// Mitsubishi GX Works2 project: 0624(BKRST_일괄리셋)   PLC: Q02/Q02H

PROGRAM MAIN
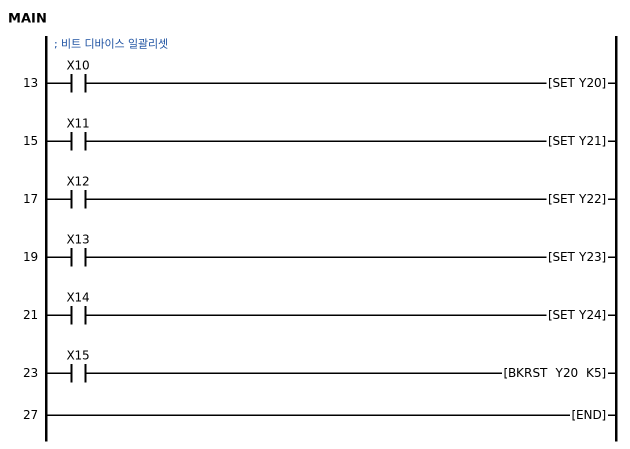
; 비트 디바이스 일괄리셋
13    LD      X10
      SET     Y20
15    LD      X11
      SET     Y21
17    LD      X12
      SET     Y22
19    LD      X13
      SET     Y23
21    LD      X14
      SET     Y24
23    LD      X15
      BKRST   Y20 K5
27    END
END_PROGRAM
